// Core §3.8b - named parameter sets kept on any I_PersistMedium: each set is
// one FB_ConfigSetDocument ('<KeyPrefix>.set<n>'), so on the file medium a set
// is a readable JSON-lines file and on the retentive medium a pooled document.
// The project picks the medium; this store is the same either way.
//
// The sets are held in volatile slots for the synchronous I_ConfigStore reads,
// read back from the medium once at start, and every saved or deleted set is
// written out. It is also this store's I_ConfigPersistence: the owning root finds
// it by __QUERYINTERFACE and drives it with every other durability provider, so
// PersistPending covers a saved set until its document is written (§3.8b), and
// a project wires nothing beyond SetConfigStore.
//
// Like every store it validates nothing and authorizes nothing (§5.6, §14); a
// set restored here is still validated by the root when somebody loads it. A set
// lost on the medium is reported by RestoreLost and is simply not listed, as
// FB_LocalConfigStore reports a rejected table.
FUNCTION_BLOCK FB_MediumConfigStore IMPLEMENTS I_ConfigStore, I_ConfigPersistence
VAR_OUTPUT
    Restored    : BOOL;   // every stored set has been read back
    RestoreLost : BOOL;   // a set the medium had, or confirmed, did not come back
    Durable     : BOOL;   // every saved and deleted set is written
END_VAR
VAR
    {attribute 'OPC.UA.DA' := '0'}
    _medium : I_PersistMedium;
    _prefix : STRING(60);
    {attribute 'OPC.UA.DA' := '0'}
    _sets   : ARRAY[1..PL_Fraktal.MAX_CONFIG_SETS] OF FB_ConfigSnapshot;
    _dirty  : ARRAY[1..PL_Fraktal.MAX_CONFIG_SETS] OF BOOL;
    // The open save. A set becomes visible only at M_SaveCommit, exactly as in
    // FB_LocalConfigStore: an aborted or refused save leaves the old set intact.
    _saveSlot : INT;
    {attribute 'OPC.UA.DA' := '0'}
    _staged   : FB_ConfigSnapshot;
    {attribute 'OPC.UA.DA' := '0'}
    _doc      : FB_ConfigSetDocument;
    _phase    : INT;
    _slot     : INT;
    _failed   : BOOL;
    _retry    : TON;
END_VAR
VAR CONSTANT
    RETRY_INTERVAL : TIME := T#10S;
END_VAR

// no cyclic body: the owning root drives M_Cyclic

// The medium and the key prefix (letters, digits, '_', '.', '-'; at most 60).
// Refused once the restore has started.
METHOD Setup : BOOL
VAR_INPUT
    Medium    : I_PersistMedium;
    KeyPrefix : STRING(60);
END_VAR
Setup := FALSE;
IF (_phase <> 0) OR (Medium = 0) OR NOT F_ValidPersistKey(Key := KeyPrefix) THEN
    RETURN;
END_IF
_medium := Medium;
_prefix := KeyPrefix;
Setup := TRUE;
END_METHOD

METHOD M_Kind : E_ConfigStore
M_Kind := E_ConfigStore.FILE_JSON;
IF _medium <> 0 THEN
    M_Kind := _medium.M_Kind();
END_IF
END_METHOD

// I_ConfigPersistence - the changed sets are already marked; a new request
// re-arms a failed write at once instead of after the retry interval.
METHOD M_Request : BOOL
_retry(IN := FALSE, PT := RETRY_INTERVAL);
_failed := FALSE;
M_Request := _medium <> 0;
END_METHOD

METHOD M_Failed : BOOL
M_Failed := _failed;
END_METHOD

// I_ConfigPersistence - read every set back once, then write each changed set.
// TRUE while the restore runs or a changed set is not yet written.
METHOD M_Cyclic : BOOL
VAR
    i    : INT;
    info : ST_ConfigSetInfo;
    seen : ST_ConfigSetInfo;
    k    : INT;
END_VAR
M_Cyclic := FALSE;
IF _medium = 0 THEN
    RETURN;
END_IF
CASE _phase OF
    0:      // restore: read slot 1 first
        _slot := 1;
        _phase := 10;
    10:
        IF _doc.M_Read(Medium := _medium, Key := _M_Key(Slot := _slot)) THEN
            _phase := 11;
        END_IF
    11:
        IF _doc.M_Poll() AND NOT _doc.Ok THEN
            // The medium could not answer: the same set is asked for again later.
            _failed := TRUE;
            _retry(IN := FALSE, PT := RETRY_INTERVAL);
            _phase := 12;
        ELSIF NOT _doc.Busy THEN
            _failed := FALSE;
            IF _doc.Lost THEN
                RestoreLost := TRUE;
            END_IF
            IF _doc.Found THEN
                IF _doc.M_Parse(Store := _sets[_slot], Info := info) THEN
                    // A set name appears once; a second copy is not listed.
                    FOR k := 1 TO _slot - 1 DO
                        IF _sets[k].M_ReadInfo(SetName := info.SetName, Info := seen) THEN
                            _sets[_slot].M_Delete(SetName := info.SetName);
                            RestoreLost := TRUE;
                        END_IF
                    END_FOR
                ELSE
                    RestoreLost := TRUE;
                END_IF
            END_IF
            IF _slot < PL_Fraktal.MAX_CONFIG_SETS THEN
                _slot := _slot + 1;
                _phase := 10;
            ELSE
                Restored := TRUE;
                _phase := 30;
            END_IF
        END_IF
    12:
        _retry(IN := TRUE, PT := RETRY_INTERVAL);
        IF _retry.Q THEN
            _retry(IN := FALSE, PT := RETRY_INTERVAL);
            _phase := 10;
        END_IF
    30:     // idle: write the first changed set
        _retry(IN := _failed, PT := RETRY_INTERVAL);
        IF NOT _failed OR _retry.Q THEN
            FOR i := 1 TO PL_Fraktal.MAX_CONFIG_SETS DO
                IF _dirty[i] AND (_phase = 30) THEN
                    _slot := i;
                    _phase := 40;
                END_IF
            END_FOR
        END_IF
    40:
        _retry(IN := FALSE, PT := RETRY_INTERVAL);
        IF _sets[_slot].M_InfoAt(Index := 1, Info := info) THEN
            IF _doc.M_Write(Medium := _medium, Key := _M_Key(Slot := _slot),
                    Store := _sets[_slot], SetName := info.SetName) THEN
                _dirty[_slot] := FALSE;     // a commit during the write marks it again
                _phase := 41;
            ELSE
                _M_WriteDone(Ok := FALSE);
            END_IF
        ELSIF _doc.M_Delete(Medium := _medium, Key := _M_Key(Slot := _slot)) THEN
            _dirty[_slot] := FALSE;
            _phase := 41;
        ELSE
            _M_WriteDone(Ok := FALSE);
        END_IF
    41:
        IF _doc.M_Poll() THEN
            _M_WriteDone(Ok := _doc.Ok);
        END_IF
ELSE
    _phase := 30;
END_CASE
// Durable only when idle: a set whose write is in flight is not yet safe.
Durable := (_phase = 30) AND NOT _failed;
FOR i := 1 TO PL_Fraktal.MAX_CONFIG_SETS DO
    IF _dirty[i] THEN
        Durable := FALSE;
    END_IF
END_FOR
M_Cyclic := NOT Durable;
END_METHOD

METHOD PRIVATE _M_WriteDone
VAR_INPUT
    Ok : BOOL;
END_VAR
IF Ok THEN
    _failed := FALSE;
ELSE
    _dirty[_slot] := TRUE;     // retried after RETRY_INTERVAL
    _failed := TRUE;
END_IF
_phase := 30;
END_METHOD

METHOD PRIVATE _M_Key : STRING(80)
VAR_INPUT
    Slot : INT;
END_VAR
_M_Key := CONCAT(_prefix, CONCAT('.set', INT_TO_STRING(Slot)));
END_METHOD

METHOD PRIVATE _M_Find : INT
VAR_INPUT
    SetName : STRING(80);
END_VAR
VAR
    i : INT;
    info : ST_ConfigSetInfo;
END_VAR
_M_Find := 0;
IF SetName = '' THEN
    RETURN;
END_IF
FOR i := 1 TO PL_Fraktal.MAX_CONFIG_SETS DO
    IF _sets[i].M_ReadInfo(SetName := SetName, Info := info) THEN
        _M_Find := i;
        RETURN;
    END_IF
END_FOR
END_METHOD

// Open a save into the slot holding this name, else a free one. Refused until
// the stored sets are back: a save then could silently replace one.
METHOD M_SaveBegin : BOOL
VAR_INPUT
    Info : ST_ConfigSetInfo;
END_VAR
VAR
    i : INT;
END_VAR
M_SaveBegin := FALSE;
_saveSlot := 0;
IF NOT Restored OR (Info.SetName = '') THEN
    RETURN;
END_IF
_saveSlot := _M_Find(SetName := Info.SetName);
IF _saveSlot = 0 THEN
    FOR i := 1 TO PL_Fraktal.MAX_CONFIG_SETS DO
        IF (_saveSlot = 0) AND (_sets[i].M_Count() = 0) THEN
            _saveSlot := i;
        END_IF
    END_FOR
END_IF
IF _saveSlot = 0 THEN
    RETURN;                     // full: refuse, never evict somebody's set
END_IF
M_SaveBegin := _staged.M_SaveBegin(Info := Info);
IF NOT M_SaveBegin THEN
    _saveSlot := 0;
END_IF
END_METHOD

METHOD M_SaveRecord : BOOL
VAR_INPUT
    Record : ST_ConfigRecord;
END_VAR
M_SaveRecord := FALSE;
IF _saveSlot = 0 THEN
    RETURN;
END_IF
M_SaveRecord := _staged.M_SaveRecord(Record := Record);
END_METHOD

METHOD M_SaveCommit : BOOL
M_SaveCommit := FALSE;
IF _saveSlot = 0 THEN
    RETURN;
END_IF
IF _staged.M_SaveCommit() THEN
    _sets[_saveSlot] := _staged;            // published in one assignment
    _dirty[_saveSlot] := TRUE;
    Durable := FALSE;
    M_SaveCommit := TRUE;
END_IF
_saveSlot := 0;
END_METHOD

METHOD M_SaveAbort : BOOL
_staged.M_SaveAbort();
_saveSlot := 0;
M_SaveAbort := TRUE;
END_METHOD

METHOD M_ReadInfo : BOOL
VAR_INPUT
    SetName : STRING(80);
END_VAR
VAR_IN_OUT
    Info : ST_ConfigSetInfo;
END_VAR
VAR
    slot : INT;
END_VAR
M_ReadInfo := FALSE;
slot := _M_Find(SetName := SetName);
IF slot > 0 THEN
    M_ReadInfo := _sets[slot].M_ReadInfo(SetName := SetName, Info := Info);
END_IF
END_METHOD

METHOD M_ReadRecord : BOOL
VAR_INPUT
    SetName : STRING(80);
    Index   : INT;
END_VAR
VAR_IN_OUT
    Record : ST_ConfigRecord;
END_VAR
VAR
    slot : INT;
END_VAR
M_ReadRecord := FALSE;
slot := _M_Find(SetName := SetName);
IF slot > 0 THEN
    M_ReadRecord := _sets[slot].M_ReadRecord(SetName := SetName, Index := Index,
        Record := Record);
END_IF
END_METHOD

METHOD M_Count : INT
VAR
    i : INT;
END_VAR
M_Count := 0;
FOR i := 1 TO PL_Fraktal.MAX_CONFIG_SETS DO
    M_Count := M_Count + _sets[i].M_Count();
END_FOR
END_METHOD

METHOD M_Delete : BOOL
VAR_INPUT
    SetName : STRING(80);
END_VAR
VAR
    slot : INT;
END_VAR
M_Delete := FALSE;
slot := _M_Find(SetName := SetName);
IF (slot = 0) OR (slot = _saveSlot) THEN
    RETURN;                     // unknown, or a save into this slot is open
END_IF
M_Delete := _sets[slot].M_Delete(SetName := SetName);
IF M_Delete THEN
    _dirty[slot] := TRUE;
    Durable := FALSE;
END_IF
END_METHOD

// Index runs over the OCCUPIED sets in slot order (1..M_Count).
METHOD M_InfoAt : BOOL
VAR_INPUT
    Index : INT;
END_VAR
VAR_IN_OUT
    Info : ST_ConfigSetInfo;
END_VAR
VAR
    i    : INT;
    seen : INT;
END_VAR
M_InfoAt := FALSE;
seen := 0;
FOR i := 1 TO PL_Fraktal.MAX_CONFIG_SETS DO
    seen := seen + _sets[i].M_Count();
    IF (seen = Index) AND (_sets[i].M_Count() = 1) THEN
        M_InfoAt := _sets[i].M_InfoAt(Index := 1, Info := Info);
        RETURN;
    END_IF
END_FOR
END_METHOD

END_FUNCTION_BLOCK

(* stored: Version 1.1.0.1, ProductVersion 3.1.4024.12
   POU FB_MediumConfigStore: Id {94397e4f-5921-4f68-a308-53092d3cb201}, SpecialFunc None
   Method Setup: Id {fa3c4957-6725-4fff-99c4-2141dc9db155}
   Method M_Kind: Id {37f0b6a6-3eaa-42e1-ab66-04a63f415fe5}
   Method M_Request: Id {d801d894-84ca-4828-82f1-4b5a54ae2f9e}
   Method M_Failed: Id {9b1d6ec2-5167-42d6-af24-2468ab86227e}
   Method M_Cyclic: Id {56cf1021-7cda-4189-9d52-95db10030de1}
   Method _M_WriteDone: Id {e9563599-02d6-4396-8b90-d3a7c94b150c}
   Method _M_Key: Id {87cdc2a0-201f-40d9-a2e3-ac710fd3d923}
   Method _M_Find: Id {ef8836d8-990e-444f-9893-3ae8639d3d0a}
   Method M_SaveBegin: Id {c90a064f-5c7a-4465-8eb4-4c925701cd2c}
   Method M_SaveRecord: Id {74357700-90c7-4abc-adfc-9a3cae20aac0}
   Method M_SaveCommit: Id {47bfaf5d-650d-4bb4-b1c5-fb0d3650fa9b}
   Method M_SaveAbort: Id {0e62814c-83e0-4f13-b511-1885b9bca27b}
   Method M_ReadInfo: Id {19eefa8a-b539-4b61-8922-2542649eddb4}
   Method M_ReadRecord: Id {76b28faf-36a7-437d-b266-9c61d00cd0ce}
   Method M_Count: Id {19a6d1e8-bcf2-4511-9830-f56db4c0e48d}
   Method M_Delete: Id {a5f898b0-099c-4903-acf6-4685410bf619}
   Method M_InfoAt: Id {a33879a7-c39e-4e74-a82e-efa0f08f5dd5} *)
